{attribute 'qualified_only'}
VAR_GLOBAL
	Data: typeStationMode;
	hmiHeader:typeHMIheader;
	
	
	//all motion rows in the station, to be inserted into the main HMI motion screen
	MotionRow: ARRAY[1..99] OF typeMotionRow;
	MotionRowBtn: ARRAY[1..99] OF typeMotionRowButtons;
	

	part: typeStationTask;
END_VAR

(* stored: Version 1.1.0.1, ProductVersion 3.1.4024.12
   GVL S5_Global: Id {a78285e0-e1c4-4163-8848-014e01ba6957} *)
